# EPICS substitutions: siteApps/EtherCat/m-epics-ecat2db/db/ecat2el3202.substitutions
file ecat2slave.template
{
	pattern {DEVICENAME}
		{EL3202}
}

file ecat2el360xel320x.template
{
	pattern {CH_ID, PDO_IDX, ESLO, EGU, PREC}
		{$(MOD_ID)-RTD1, 0, 0.01, °C, 2}
		{$(MOD_ID)-RTD2, 1, 0.01, °C, 2}
}
